TYPE ST_DiscreteValveDefaultParameters :
STRUCT
	nFeedback : E_DiscreteValveFeedbackMode;
END_STRUCT
END_TYPE

(* stored: Version 1.1.0.1, ProductVersion 3.1.4024.10
   DUT ST_DiscreteValveDefaultParameters: Id {91238d3e-c396-45dc-abc4-16aa2710a625} *)
